Staubli VAL3: page_program.dtx

num nTime = 1
num nKey
num nRefresh
public num nPage
num nIndex
num nView
num nSelected
public string sItems
string sMessage
string sMenu
string sEvent
string sList
string sMenu8[8]
bool bButton[8]
string sProgType
num nProgID
